% RSLogix 500 project Project_4.RSS, saved by version 8.30.00.16 %
PROJECT "UNTITLED"    % processor: Bul.1763 MicroLogix 1100 Series B %

PROGRAM FILES
  LAD 2   3 rungs
  LAD 3 "IO"  8 rungs  % Input/Output %
  LAD 4 "LOGIC"  24 rungs  % Logic %

DATA FILES
  O0 OUTPUT  4 elements
  I1 INPUT  6 elements
  S2 STATUS  66 elements
  B3 BINARY  32 elements
  T4 TIMER  3 elements
  C5 COUNTER  1 elements
  R6 CONTROL  1 elements
  N7 INTEGER  2 elements
  F8 FLOAT  1 elements

LADDER 2
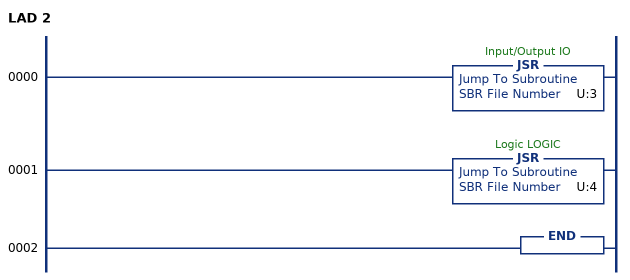
% Rung: 0 %
SOR JSR U:3 EOR
%   U:3  IO  "Input/Output" %
% Rung: 1 %
SOR JSR U:4 EOR
%   U:4  LOGIC  "Logic" %
% Rung: 2 %
SOR END EOR

LADDER 3 "IO"    % Input/Output %
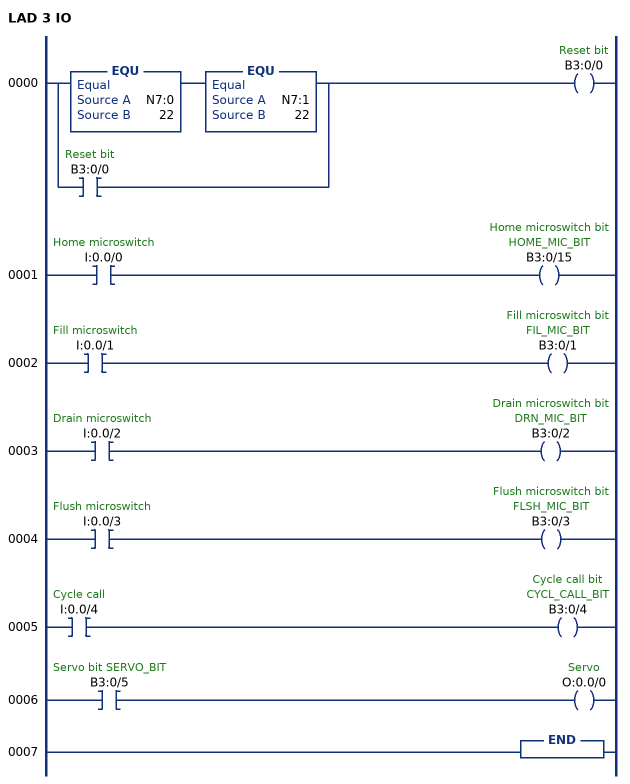
% Rung: 0 %
SOR BST EQU N7:0 22 EQU N7:1 22 NXB XIC B3:0/0 BND OTE B3:0/0 EOR
%   B3:0/0  "Reset bit" %
% Rung: 1 %
SOR XIC I:0.0/0 OTE B3:0/15 EOR
%   I:0.0/0  "Home microswitch" %
%   B3:0/15  HOME_MIC_BIT  "Home microswitch bit" %
% Rung: 2 %
SOR XIC I:0.0/1 OTE B3:0/1 EOR
%   I:0.0/1  "Fill microswitch" %
%   B3:0/1  FIL_MIC_BIT  "Fill microswitch bit" %
% Rung: 3 %
SOR XIC I:0.0/2 OTE B3:0/2 EOR
%   I:0.0/2  "Drain microswitch" %
%   B3:0/2  DRN_MIC_BIT  "Drain microswitch bit" %
% Rung: 4 %
SOR XIC I:0.0/3 OTE B3:0/3 EOR
%   I:0.0/3  "Flush microswitch" %
%   B3:0/3  FLSH_MIC_BIT  "Flush microswitch bit" %
% Rung: 5 %
SOR XIC I:0.0/4 OTE B3:0/4 EOR
%   I:0.0/4  "Cycle call" %
%   B3:0/4  CYCL_CALL_BIT  "Cycle call bit" %
% Rung: 6 %
SOR XIC B3:0/5 OTE O:0.0/0 EOR
%   B3:0/5  SERVO_BIT  "Servo bit" %
%   O:0.0/0  "Servo" %
% Rung: 7 %
SOR END EOR

LADDER 4 "LOGIC"    % Logic %
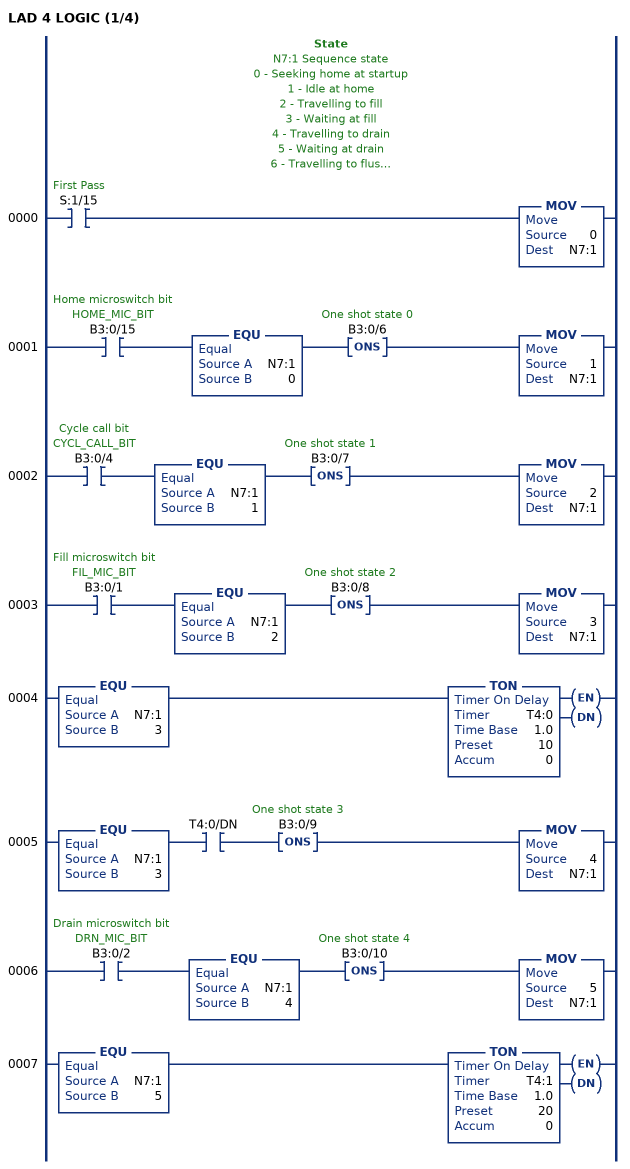
% Rung: 0 %
% TITLE: State %
% N7:1 Sequence state
% 0 - Seeking home at startup
% 1 - Idle at home
% 2 - Travelling to fill
% 3 - Waiting at fill
% 4 - Travelling to drain
% 5 - Waiting at drain
% 6 - Travelling to flush
% 7 - Waiting at flush
% 8 - Returning home
% 9 - Abort initiated, wait for home switch to open %
SOR XIC S:1/15 MOV 0 N7:1 EOR
%   S:1/15  "First Pass" %
% Rung: 1 %
SOR XIC B3:0/15 EQU N7:1 0 ONS B3:0/6 MOV 1 N7:1 EOR
%   B3:0/15  HOME_MIC_BIT  "Home microswitch bit" %
%   B3:0/6  "One shot state 0" %
% Rung: 2 %
SOR XIC B3:0/4 EQU N7:1 1 ONS B3:0/7 MOV 2 N7:1 EOR
%   B3:0/4  CYCL_CALL_BIT  "Cycle call bit" %
%   B3:0/7  "One shot state 1" %
% Rung: 3 %
SOR XIC B3:0/1 EQU N7:1 2 ONS B3:0/8 MOV 3 N7:1 EOR
%   B3:0/1  FIL_MIC_BIT  "Fill microswitch bit" %
%   B3:0/8  "One shot state 2" %
% Rung: 4 %
SOR EQU N7:1 3 TON T4:0 1.0 10 0 EOR
% Rung: 5 %
SOR EQU N7:1 3 XIC T4:0/DN ONS B3:0/9 MOV 4 N7:1 EOR
%   B3:0/9  "One shot state 3" %
% Rung: 6 %
SOR XIC B3:0/2 EQU N7:1 4 ONS B3:0/10 MOV 5 N7:1 EOR
%   B3:0/2  DRN_MIC_BIT  "Drain microswitch bit" %
%   B3:0/10  "One shot state 4" %
% Rung: 7 %
SOR EQU N7:1 5 TON T4:1 1.0 20 0 EOR

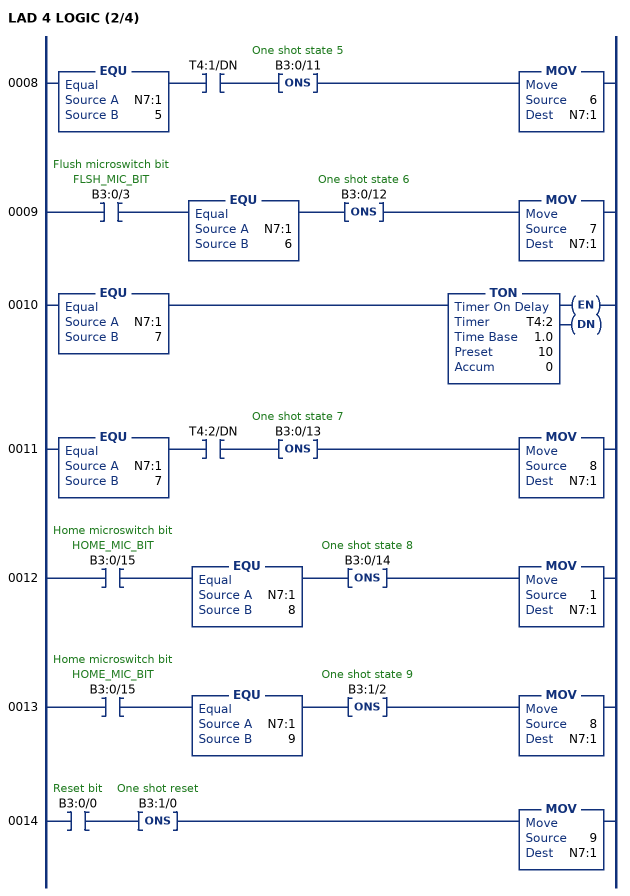
% Rung: 8 %
SOR EQU N7:1 5 XIC T4:1/DN ONS B3:0/11 MOV 6 N7:1 EOR
%   B3:0/11  "One shot state 5" %
% Rung: 9 %
SOR XIC B3:0/3 EQU N7:1 6 ONS B3:0/12 MOV 7 N7:1 EOR
%   B3:0/3  FLSH_MIC_BIT  "Flush microswitch bit" %
%   B3:0/12  "One shot state 6" %
% Rung: 10 %
SOR EQU N7:1 7 TON T4:2 1.0 10 0 EOR
% Rung: 11 %
SOR EQU N7:1 7 XIC T4:2/DN ONS B3:0/13 MOV 8 N7:1 EOR
%   B3:0/13  "One shot state 7" %
% Rung: 12 %
SOR XIC B3:0/15 EQU N7:1 8 ONS B3:0/14 MOV 1 N7:1 EOR
%   B3:0/15  HOME_MIC_BIT  "Home microswitch bit" %
%   B3:0/14  "One shot state 8" %
% Rung: 13 %
SOR XIC B3:0/15 EQU N7:1 9 ONS B3:1/2 MOV 8 N7:1 EOR
%   B3:0/15  HOME_MIC_BIT  "Home microswitch bit" %
%   B3:1/2  "One shot state 9" %
% Rung: 14 %
SOR XIC B3:0/0 ONS B3:1/0 MOV 9 N7:1 EOR
%   B3:0/0  "Reset bit" %
%   B3:1/0  "One shot reset" %

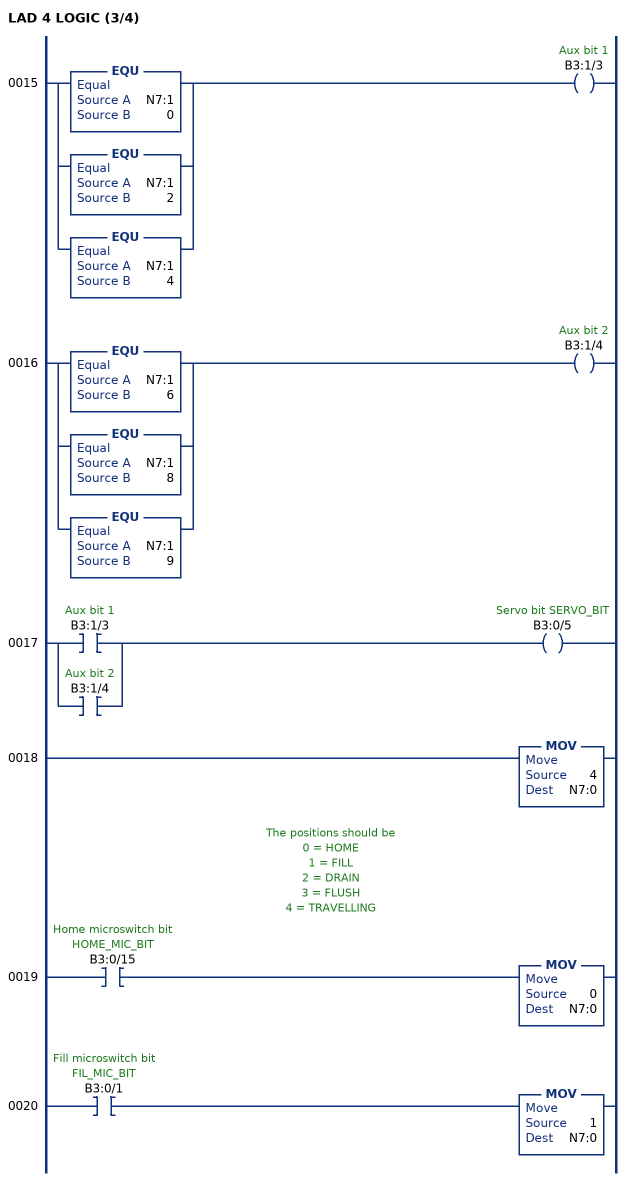
% Rung: 15 %
SOR BST EQU N7:1 0 NXB BST EQU N7:1 2 NXB EQU N7:1 4 BND BND OTE B3:1/3 EOR
%   B3:1/3  "Aux bit 1" %
% Rung: 16 %
SOR BST EQU N7:1 6 NXB BST EQU N7:1 8 NXB EQU N7:1 9 BND BND OTE B3:1/4 EOR
%   B3:1/4  "Aux bit 2" %
% Rung: 17 %
SOR BST XIC B3:1/3 NXB XIC B3:1/4 BND OTE B3:0/5 EOR
%   B3:1/3  "Aux bit 1" %
%   B3:1/4  "Aux bit 2" %
%   B3:0/5  SERVO_BIT  "Servo bit" %
% Rung: 18 %
SOR MOV 4 N7:0 EOR
% Rung: 19 %
% The positions should be
% 0 = HOME
% 1 = FILL
% 2 = DRAIN
% 3 = FLUSH
% 4 = TRAVELLING %
SOR XIC B3:0/15 MOV 0 N7:0 EOR
%   B3:0/15  HOME_MIC_BIT  "Home microswitch bit" %
% Rung: 20 %
SOR XIC B3:0/1 MOV 1 N7:0 EOR
%   B3:0/1  FIL_MIC_BIT  "Fill microswitch bit" %

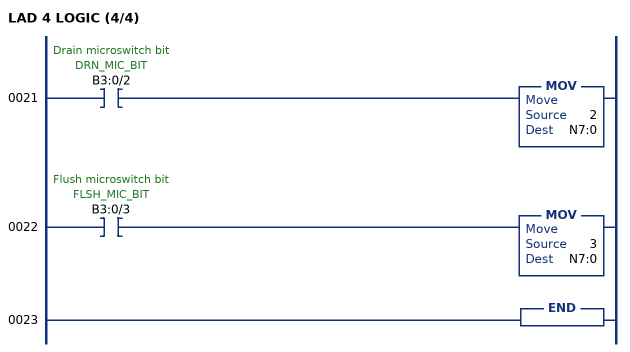
% Rung: 21 %
SOR XIC B3:0/2 MOV 2 N7:0 EOR
%   B3:0/2  DRN_MIC_BIT  "Drain microswitch bit" %
% Rung: 22 %
SOR XIC B3:0/3 MOV 3 N7:0 EOR
%   B3:0/3  FLSH_MIC_BIT  "Flush microswitch bit" %
% Rung: 23 %
SOR END EOR

DATA TABLE (non-zero values as saved)
DATA B3
% B3:0 % 0X8020 0X0008 0X0000 0X0000 0X0000 0X0000 0X0000 0X0000 0X0000 0X0000
DATA T4
% .PRE .ACC %
% T4:0 % 10 0
% T4:1 % 20 0
% T4:2 % 10 0
DATA N7
% N7:0 % 0 2
